(* IEC 61131-3 sources: Elmo_Master/Lasal_PRG/Elmo_EtherCAT_Test_4Axis/Class/EtherCATSlot_Hub_Base, 1 file *)

(* ---- EtherCATSlot_Hub_Base.st ---- *)
(*!
<Class
	Name               = "EtherCATSlot_Hub_Base"
	Revision           = "1.1"
	RealtimeTask       = "false"
	CyclicTask         = "false"
	BackgroundTask     = "false"
	Sigmatek           = "true"
	OSInterface        = "false"
	HighPriority       = "false"
	Automatic          = "false"
	UpdateMode         = "Prescan"
	IconPath           = ".\Class\EtherCAT.ico"
	SharedCommandTable = "true"
	Objectsize         = "(494,120)">
	<Channels>
		<Server Name="ClassSvr" Visualized="false" Initialize="false" WriteProtected="true" Retentive="false" Comment="Connect an EtherCATSlot Slave."/>
		<Client Name="SplitterPlace" Required="true" Internal="false" Comment="Place of this splitter."/>
		<Client Name="toNextEtherCAT" Required="true" Internal="false" Comment="Connect to first server of Ethercat master."/>
	</Channels>
	<RevDoku>
		<Owner Company="Sigmatek" Author="LanSte"/>
		<Dokumentation Revision="1.1" Date="2026-04-10" Author="LanSte" Company="Sigmatek" Description="Special: Set property flag &quot;Hidden&quot; of class, since this is an internal class."/>
		<Dokumentation Revision="1.0" Date="01.12.2023" Author="LanSte" Company="Sigmatek" Description="First library version."/>
	</RevDoku>
	<AdditionalData>
		<Entry Name="Hidden" Value="true"/>
	</AdditionalData>
</Class>
*)
EtherCATSlot_Hub_Base : CLASS
  //Servers:
	ClassSvr 	: SvrChCmd_DINT;
  //Clients:
	toNextEtherCAT 	: CltChCmd_t_e_VaranErrors;
	SplitterPlace 	: CltCh_DINT;
  //Variables:
  //Functions:

	FUNCTION VIRTUAL GLOBAL ClassSvr::NewInst
		VAR_INPUT
			pPara 	: ^CmdStruct;
			pResult 	: ^results;
		END_VAR
		VAR_OUTPUT
			ret_code 	: iprStates;
		END_VAR;
  //Tables:
	FUNCTION @STD
		VAR_OUTPUT
			ret_code	: CONFSTATES;
		END_VAR;
	FUNCTION GLOBAL TAB @CT_;
END_CLASS;

FUNCTION VIRTUAL GLOBAL EtherCATSlot_Hub_Base::ClassSvr::NewInst
	VAR_INPUT
		pPara 	: ^CmdStruct;
		pResult 	: ^results;
	END_VAR
	VAR_OUTPUT
		ret_code 	: iprStates;
	END_VAR

  // use last parameter for port number
  pPara^.aPara[MAXCMDPARA-1] := SplitterPlace;

	ret_code := toNextEtherCAT.NewInst(pPara, pResult);

END_FUNCTION
